(* IEC 61131-3 sources: Industry-PLC-LLM/data/PLCBEAD_repo/PLCBEAD_PLCEmbed-main/PLC-BEAD/Source/GEB/GOLD, 1 file *)

(* ---- GOLD.ST ---- *)
FUNCTION GOLD:REAL

	VAR_INPUT
		X :	REAL;
	END_VAR

	GOLD := (X + SQRT(X*X + 4.0)) * 0.5;

END_FUNCTION

PROGRAM program0
  VAR
   	X :	REAL;
    LocalOUT  : REAL;
  END_VAR

  LocalOUT := GOLD(X);
END_PROGRAM
